(* PLC project v0.6.02_RefactorGateAndTest.project, CODESYS CODESYS V3.5 SP19 Patch 1 *)
(* stored: creationDateTime 2026-08-11T18:19:14.798534, modificationDateTime 2026-08-11T18:19:14.798534 *)

(* ═══════════════════════════════════════════════════════════════ ⚙️ ST_BucketConfig — Configuration des offsets du benne ─────────────────────────────────────────────────────────────── 📄 Doc métier : DOC/AF/AF_Partie-10_Fonction_Winch/FB_Bucket_v1.0.md §4.A ═══════════════════════════════════════════════════════════════ *)
TYPE ST_BucketConfig : STRUCT
  OffsetOpenM : REAL;  (* Écart M1/M2 en mètres benne ouvert *)
  OffsetCloseM : REAL;  (* Écart M1/M2 en mètres benne fermé *)
  CoherenceLimitM : REAL;  (* Seuil de détection d'incohérence au boot *)
  CloseAnticipationM : REAL := 1;  (* 🆕 2026-08-07 (20) — retour terrain, demande client : inertie mécanique du benne (M2 continue sur sa lancée après coupure StartStop) -- couper la commande EN AVANCE de la cible pour que l'arrêt réel (après coast-down) tombe proche du vrai offset, au lieu de dépasser. Anticipation distincte par sens (fermeture/ouverture ont des inerties différentes selon retour terrain). Coupe la commande de fermeture 1m avant OffsetCloseM *)
  OpenAnticipationM : REAL := 1.3;  (* Coupe la commande d'ouverture 1.3m avant OffsetOpenM *)
END_STRUCT;
END_TYPE
